(* PLC project EPEC_CU1.project, CODESYS V3.5 SP19, author XXXX *)
(* stored: creationDateTime 2026-03-19T14:01:24.4396503+02:00, modificationDateTime 2026-03-19T14:01:24.4396503+02:00, organization XXXX *)

(* This PRG contains non safety-related code. The following attribute is autogenerated. Do not remove. *)
{attribute 'location' := '16#800'}
PROGRAM Main

                    
                  
END_PROGRAM

(* This PRG contains non safety-related code. The following attribute is autogenerated. Do not remove. *)
{attribute 'location' := '16#800'}
PROGRAM MainInit
  VAR_OUTPUT
    o_MainInitReady : BOOL := FALSE;
  END_VAR

                    o_MainInitReady := TRUE;
                  
END_PROGRAM

CONFIGURATION Device
  RESOURCE Application ON PLC
    TASK NonSafePRG_TASK(INTERVAL := T#10ms, PRIORITY := 1);
    PROGRAM PLC_PRG WITH NonSafePRG_TASK : PLC_PRG;
  END_RESOURCE
END_CONFIGURATION
